// TIA Portal V17 export
// export: Created 2024-09-03T21:55:01.8122438Z, ExportSetting WithDefaults, DisplayName Totally Integrated Automation Portal, DisplayVersion V17 Update 7, DisplayName TIA Portal Openness, DisplayVersion V17 Update 7, DisplayName TIA Portal Version Control Interface, DisplayVersion V17, DisplayName SINAMICS Startdrive Advanced, DisplayVersion V17 SP2, DisplayName SINAMICS Startdrive G110M, G120, G120C, G120D, G120P, G115D, DisplayVersion V17 SP2, DisplayName SINAMICS Startdrive G130, G150, S120, S150, SINAMICS MV, S210, DisplayVersion V17 SP2, DisplayName STEP 7 Professional, DisplayVersion V17 Update 7, DisplayName STEP 7 Safety, DisplayVersion V17 Update 6, DisplayName WinCC Advanced / Unified PC, DisplayVersion V17 Update 7
DATA_BLOCK "DB_IJCoreMain"   // DB1000
VERSION : 0.1
// stored: AutoNumber false, DBAccessibleFromOPCUA true, DBAccessibleFromWebserver true, InstanceOfName IJCoreMain, InstanceOfType FB
"IJCoreMain"
   // VAR
   //    Enable : Bool := true;
   //    Mode : UInt := 1;
   //    Indicator : Int;
   //    AlarmReset : Bool;
   //    AWAKE_SIGNAL { S7_SetPoint := 'True'} : "AWAKE_SIGNAL";
   //    MSG : Array[1..20] of "IJCoreMessageProcotol";
   //    NFP { S7_SetPoint := 'True'} : Array[1..4] of String[30];
   // END_VAR
BEGIN
END_DATA_BLOCK
